PROGRAM NO
VAR
	Obj : ITcoObject;
	Structure : TcoStruct;
END_VAR

END_PROGRAM

(* stored: Version 1.1.0.1
   POU NO: Id {380c2f10-c4c6-0df0-0cc6-318b9b23bdbf}, SpecialFunc None *)
